(* Logix 5000 project; controller cal1632 1756-L62 rev 16.20; software revision 16.05; part 57 of 61 *)
(* tags used below, declared in another part *)
   FAULT : BOOL;
   HMI : BOOL;
   p01r09_pb_global_reset : BOOL;
   p29_di_wdr_turret : acs800_di_normal;
   p29r15_wdra_active : BOOL;
   p29r16_wdrb_active : BOOL;
   p29r20 : routine;
   p29r20_timer_warning : TIMER[4];
   p30_di_pin_1 : BOOL;
   p30_di_pin_2 : BOOL;
   p30_di_pin_3 : BOOL;
   p30_di_pin_4 : BOOL;
   p30_di_pin_5 : BOOL;
   p30_di_pin_6 : BOOL;
   p30_di_pin_7 : BOOL;
   p30_di_pin_8 : BOOL;
   p30_di_retraction_down_ls : BOOL;
   p30_di_retraction_up_ls : BOOL;
   p30_di_rotation_fault : BOOL;
   p30_di_ss_close : BOOL;
   p30_di_ss_open : BOOL;
   p30_dint_to_hmi : DINT[16];
   p30_do_retract_motion : BOOL;
   p30_do_rotation_fwd : BOOL;
   p30_do_rotation_rev : BOOL;
   p30r01 : routine;
   p30r02 : routine;
   p30r02_fault_exists : BOOL;
   p30r02_timer_fault : TIMER[4];
   p30r02_timer_warning : TIMER[4];
   p30r02_unack_fault : BOOL;
   p30r02_unack_warning : BOOL;
   p30r02_warning_exists : BOOL;
   p30r03 : routine;
   p30r03_timer_fault : TIMER[4];
   p30r03_timer_warning : TIMER[4];
   p30r04 : routine;
   p30r04_timer_fault : TIMER[4];
   p30r04_timer_warning : TIMER[4];
   p30r05 : routine;
   p30r05_timer_fault : TIMER[4];
   p30r05_timer_warning : TIMER[4];
   p30r06 : routine;
   p30r07 : routine;
   p30r08 : routine;
   p30r09 : routine;
   p30r10 : routine;
   RETACTION_DELAY_TIMER : TIMER;
   RETRACTION_DELAY_TIMER_2 : TIMER;
(* P29_Winder, continued *)

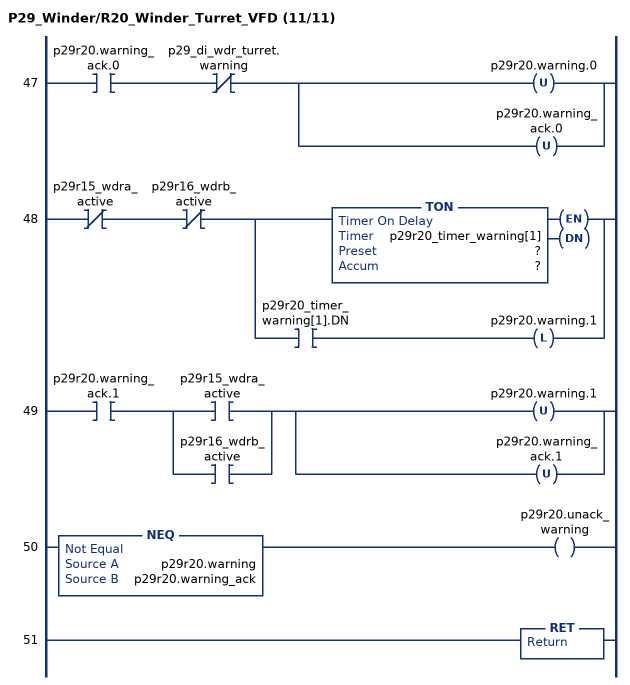
   [picture p1161: P29_Winder/R20_Winder_Turret_VFD rungs 47-51]
   47: XIC(p29r20.warning_ack.0)XIO(p29_di_wdr_turret.warning)[OTU(p29r20.warning.0) ,OTU(p29r20.warning_ack.0) ];
   48: XIO(p29r15_wdra_active)XIO(p29r16_wdrb_active)[TON(p29r20_timer_warning[1],?,?) ,XIC(p29r20_timer_warning[1].DN) OTL(p29r20.warning.1) ];
   49: XIC(p29r20.warning_ack.1)[XIC(p29r15_wdra_active) ,XIC(p29r16_wdrb_active) ][OTU(p29r20.warning.1) ,OTU(p29r20.warning_ack.1) ];
   50: NEQ(p29r20.warning,p29r20.warning_ack)OTE(p29r20.unack_warning);
   51: RET();
END_ROUTINE
END_PROGRAM

PROGRAM P30_Retraction_System   (* main routine R01_Main *)

ROUTINE R01_Main   (* ladder *)
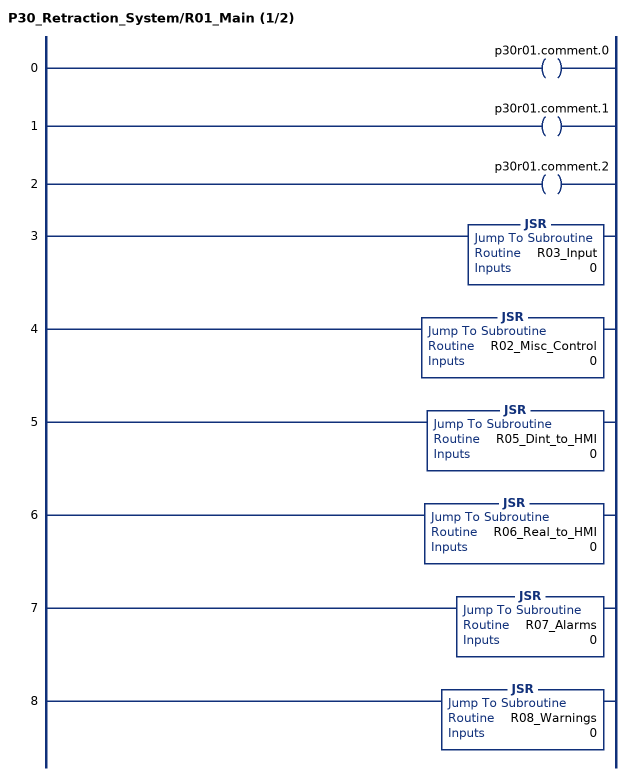
   0: OTE(p30r01.comment.0);
   1: OTE(p30r01.comment.1);
   2: OTE(p30r01.comment.2);
   3: JSR(R03_Input,0);
   4: JSR(R02_Misc_Control,0);
   5: JSR(R05_Dint_to_HMI,0);
   6: JSR(R06_Real_to_HMI,0);
   7: JSR(R07_Alarms,0);
   8: JSR(R08_Warnings,0);
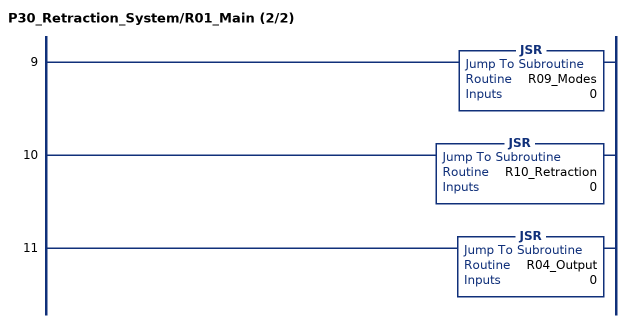
   9: JSR(R09_Modes,0);
   10: JSR(R10_Retraction,0);
   11: JSR(R04_Output,0);
END_ROUTINE

ROUTINE R02_Misc_Control   (* ladder *)
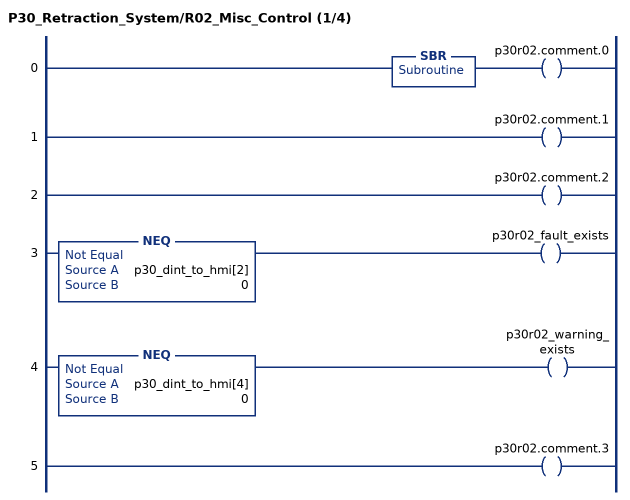
   0: SBR()OTE(p30r02.comment.0);
   1: OTE(p30r02.comment.1);
   2: OTE(p30r02.comment.2);
   3: NEQ(p30_dint_to_hmi[2],0)OTE(p30r02_fault_exists);
   4: NEQ(p30_dint_to_hmi[4],0)OTE(p30r02_warning_exists);
   5: OTE(p30r02.comment.3);
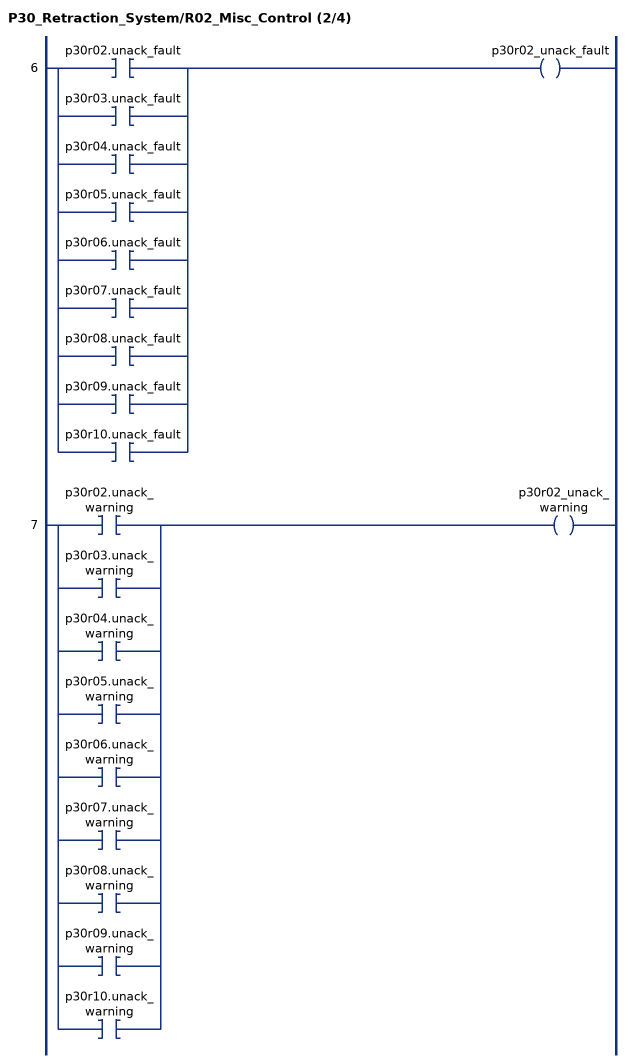
   6: [XIC(p30r02.unack_fault) ,XIC(p30r03.unack_fault) ,XIC(p30r04.unack_fault) ,XIC(p30r05.unack_fault) ,XIC(p30r06.unack_fault) ,XIC(p30r07.unack_fault) ,XIC(p30r08.unack_fault) ,XIC(p30r09.unack_fault) ,XIC(p30r10.unack_fault) ]OTE(p30r02_unack_fault);
   7: [XIC(p30r02.unack_warning) ,XIC(p30r03.unack_warning) ,XIC(p30r04.unack_warning) ,XIC(p30r05.unack_warning) ,XIC(p30r06.unack_warning) ,XIC(p30r07.unack_warning) ,XIC(p30r08.unack_warning) ,XIC(p30r09.unack_warning) ,XIC(p30r10.unack_warning) ]OTE(p30r02_unack_warning);
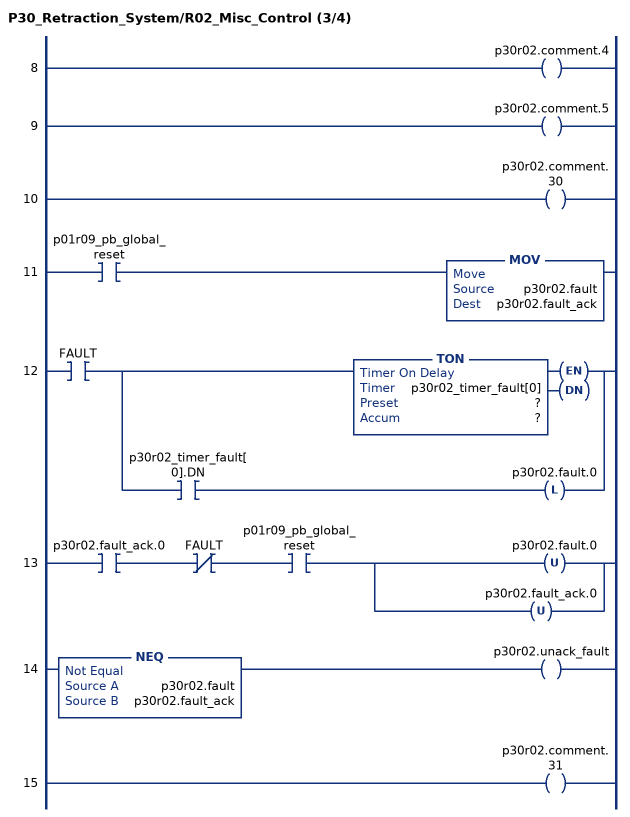
   8: OTE(p30r02.comment.4);
   9: OTE(p30r02.comment.5);
   10: OTE(p30r02.comment.30);
   11: XIC(p01r09_pb_global_reset)MOV(p30r02.fault,p30r02.fault_ack);
   12: XIC(FAULT)[TON(p30r02_timer_fault[0],?,?) ,XIC(p30r02_timer_fault[0].DN) OTL(p30r02.fault.0) ];
   13: XIC(p30r02.fault_ack.0)XIO(FAULT)XIC(p01r09_pb_global_reset)[OTU(p30r02.fault.0) ,OTU(p30r02.fault_ack.0) ];
   14: NEQ(p30r02.fault,p30r02.fault_ack)OTE(p30r02.unack_fault);
   15: OTE(p30r02.comment.31);
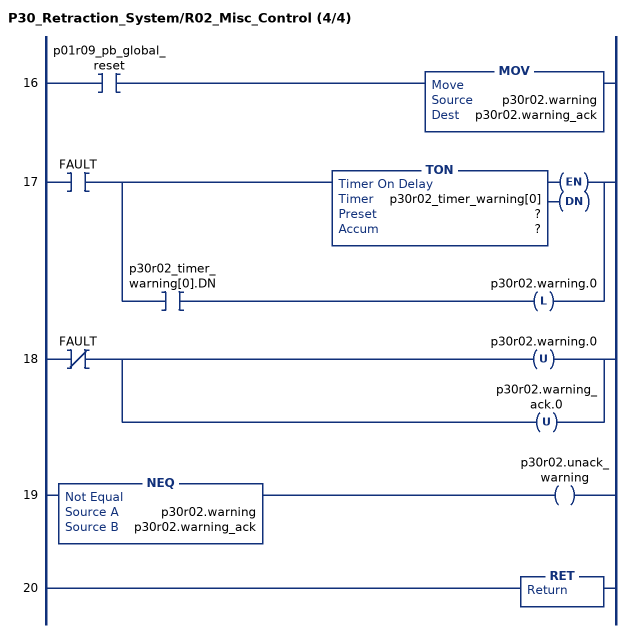
   16: XIC(p01r09_pb_global_reset)MOV(p30r02.warning,p30r02.warning_ack);
   17: XIC(FAULT)[TON(p30r02_timer_warning[0],?,?) ,XIC(p30r02_timer_warning[0].DN) OTL(p30r02.warning.0) ];
   18: XIO(FAULT)[OTU(p30r02.warning.0) ,OTU(p30r02.warning_ack.0) ];
   19: NEQ(p30r02.warning,p30r02.warning_ack)OTE(p30r02.unack_warning);
   20: RET();
END_ROUTINE

ROUTINE R03_Input   (* ladder *)
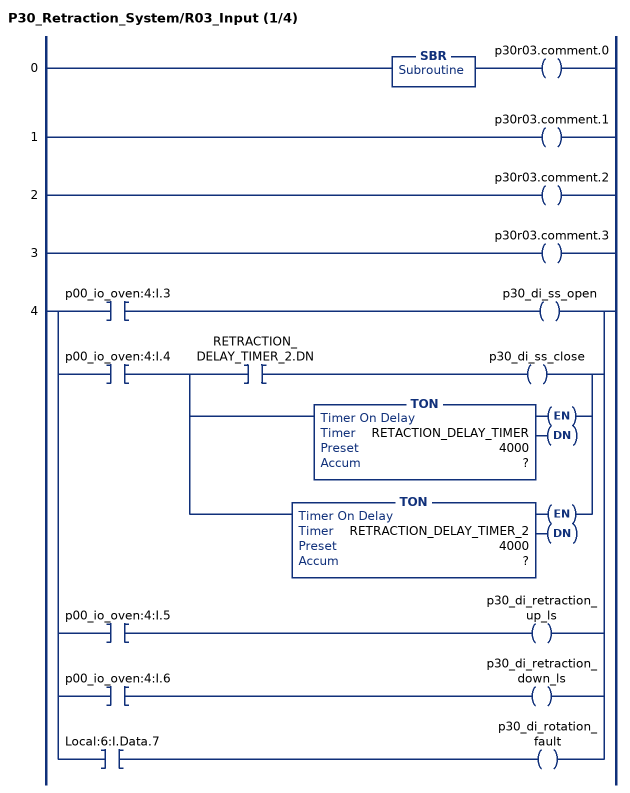
   0: SBR()OTE(p30r03.comment.0);
   1: OTE(p30r03.comment.1);
   2: OTE(p30r03.comment.2);
   3: OTE(p30r03.comment.3);
   4: [XIC(p00_io_oven:4:I.3) OTE(p30_di_ss_open) ,XIC(p00_io_oven:4:I.4) [XIC(RETRACTION_DELAY_TIMER_2.DN) OTE(p30_di_ss_close) ,TON(RETACTION_DELAY_TIMER,?,?) ,TON(RETRACTION_DELAY_TIMER_2,?,?) ] ,XIC(p00_io_oven:4:I.5) OTE(p30_di_retraction_up_ls) ,XIC(p00_io_oven:4:I.6) OTE(p30_di_retraction_down_ls) ,XIC(Local:6:I.Data.7) OTE(p30_di_rotation_fault) ];
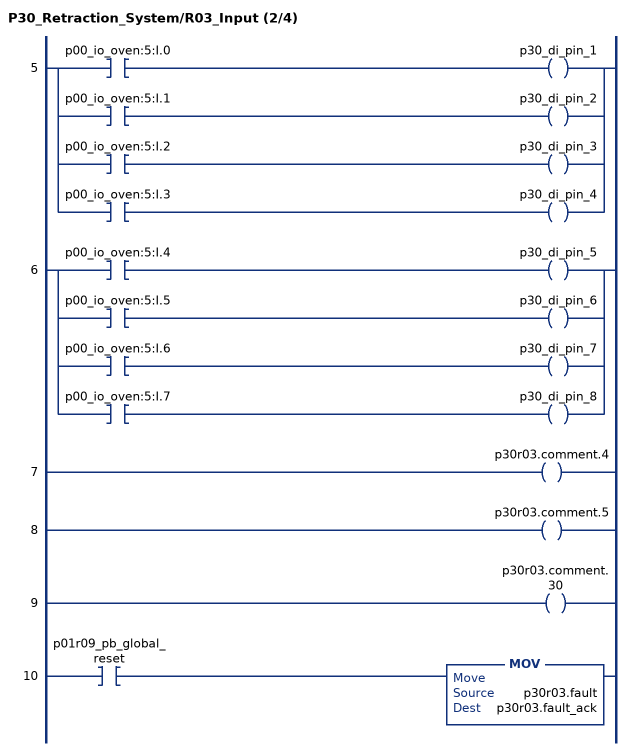
   5: [XIC(p00_io_oven:5:I.0) OTE(p30_di_pin_1) ,XIC(p00_io_oven:5:I.1) OTE(p30_di_pin_2) ,XIC(p00_io_oven:5:I.2) OTE(p30_di_pin_3) ,XIC(p00_io_oven:5:I.3) OTE(p30_di_pin_4) ];
   6: [XIC(p00_io_oven:5:I.4) OTE(p30_di_pin_5) ,XIC(p00_io_oven:5:I.5) OTE(p30_di_pin_6) ,XIC(p00_io_oven:5:I.6) OTE(p30_di_pin_7) ,XIC(p00_io_oven:5:I.7) OTE(p30_di_pin_8) ];
   7: OTE(p30r03.comment.4);
   8: OTE(p30r03.comment.5);
   9: OTE(p30r03.comment.30);
   10: XIC(p01r09_pb_global_reset)MOV(p30r03.fault,p30r03.fault_ack);
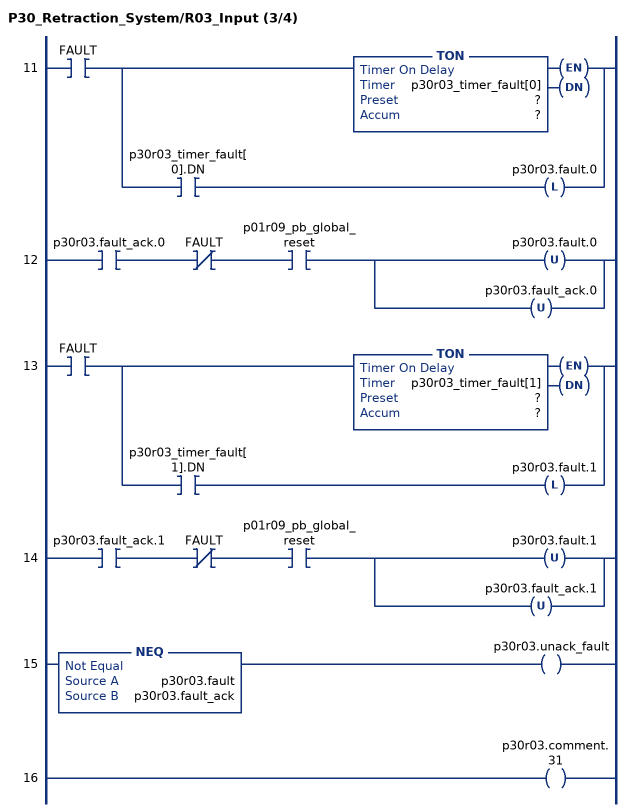
   11: XIC(FAULT)[TON(p30r03_timer_fault[0],?,?) ,XIC(p30r03_timer_fault[0].DN) OTL(p30r03.fault.0) ];
   12: XIC(p30r03.fault_ack.0)XIO(FAULT)XIC(p01r09_pb_global_reset)[OTU(p30r03.fault.0) ,OTU(p30r03.fault_ack.0) ];
   13: XIC(FAULT)[TON(p30r03_timer_fault[1],?,?) ,XIC(p30r03_timer_fault[1].DN) OTL(p30r03.fault.1) ];
   14: XIC(p30r03.fault_ack.1)XIO(FAULT)XIC(p01r09_pb_global_reset)[OTU(p30r03.fault.1) ,OTU(p30r03.fault_ack.1) ];
   15: NEQ(p30r03.fault,p30r03.fault_ack)OTE(p30r03.unack_fault);
   16: OTE(p30r03.comment.31);
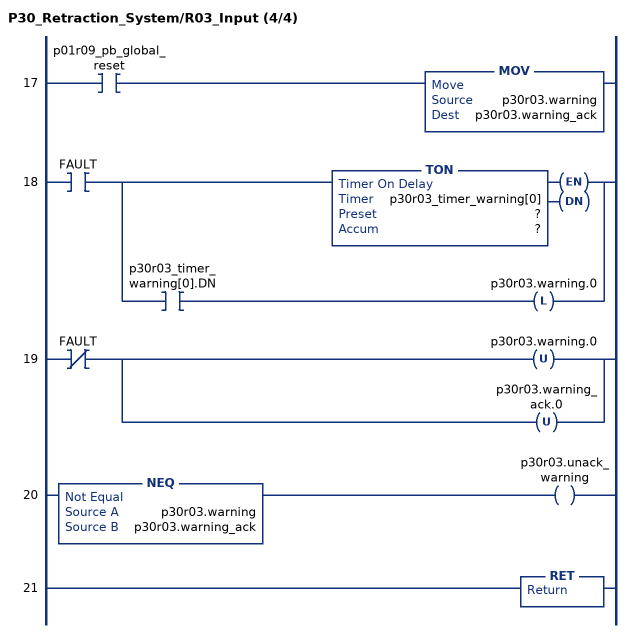
   17: XIC(p01r09_pb_global_reset)MOV(p30r03.warning,p30r03.warning_ack);
   18: XIC(FAULT)[TON(p30r03_timer_warning[0],?,?) ,XIC(p30r03_timer_warning[0].DN) OTL(p30r03.warning.0) ];
   19: XIO(FAULT)[OTU(p30r03.warning.0) ,OTU(p30r03.warning_ack.0) ];
   20: NEQ(p30r03.warning,p30r03.warning_ack)OTE(p30r03.unack_warning);
   21: RET();
END_ROUTINE

ROUTINE R04_Output   (* ladder *)
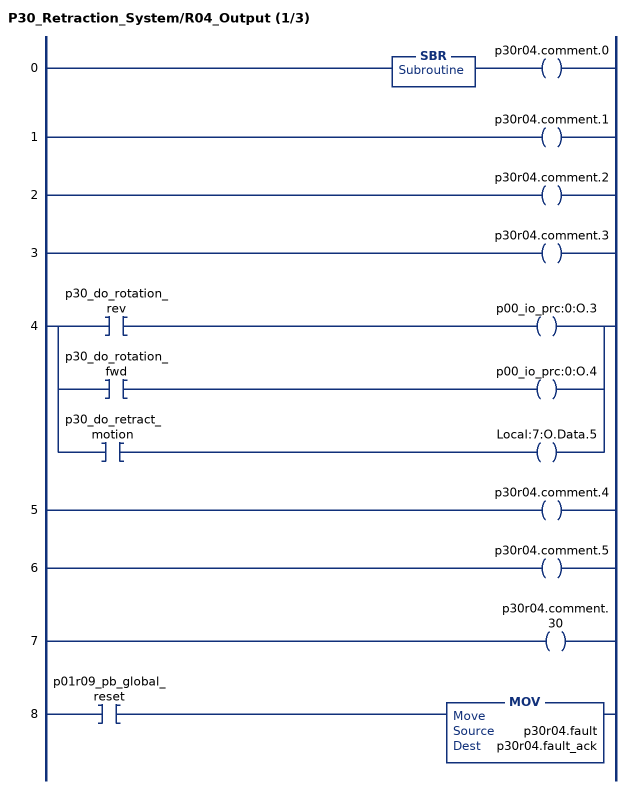
   0: SBR()OTE(p30r04.comment.0);
   1: OTE(p30r04.comment.1);
   2: OTE(p30r04.comment.2);
   3: OTE(p30r04.comment.3);
   4: [XIC(p30_do_rotation_rev) OTE(p00_io_prc:0:O.3) ,XIC(p30_do_rotation_fwd) OTE(p00_io_prc:0:O.4) ,XIC(p30_do_retract_motion) OTE(Local:7:O.Data.5) ];
   5: OTE(p30r04.comment.4);
   6: OTE(p30r04.comment.5);
   7: OTE(p30r04.comment.30);
   8: XIC(p01r09_pb_global_reset)MOV(p30r04.fault,p30r04.fault_ack);
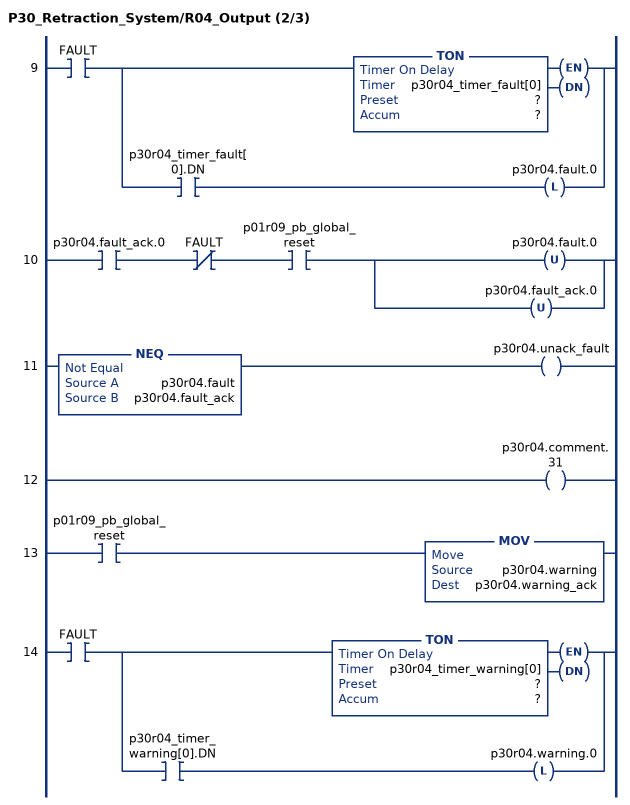
   9: XIC(FAULT)[TON(p30r04_timer_fault[0],?,?) ,XIC(p30r04_timer_fault[0].DN) OTL(p30r04.fault.0) ];
   10: XIC(p30r04.fault_ack.0)XIO(FAULT)XIC(p01r09_pb_global_reset)[OTU(p30r04.fault.0) ,OTU(p30r04.fault_ack.0) ];
   11: NEQ(p30r04.fault,p30r04.fault_ack)OTE(p30r04.unack_fault);
   12: OTE(p30r04.comment.31);
   13: XIC(p01r09_pb_global_reset)MOV(p30r04.warning,p30r04.warning_ack);
   14: XIC(FAULT)[TON(p30r04_timer_warning[0],?,?) ,XIC(p30r04_timer_warning[0].DN) OTL(p30r04.warning.0) ];
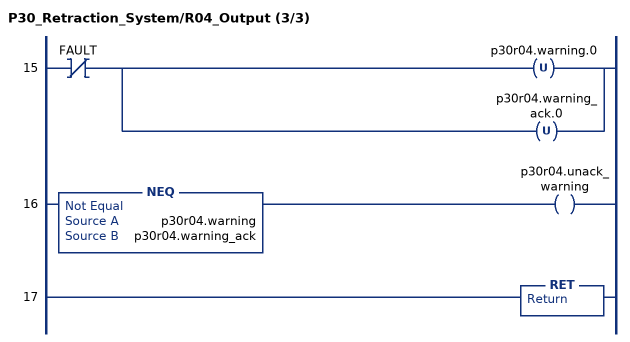
   15: XIO(FAULT)[OTU(p30r04.warning.0) ,OTU(p30r04.warning_ack.0) ];
   16: NEQ(p30r04.warning,p30r04.warning_ack)OTE(p30r04.unack_warning);
   17: RET();
END_ROUTINE

ROUTINE R05_Dint_to_HMI   (* ladder *)
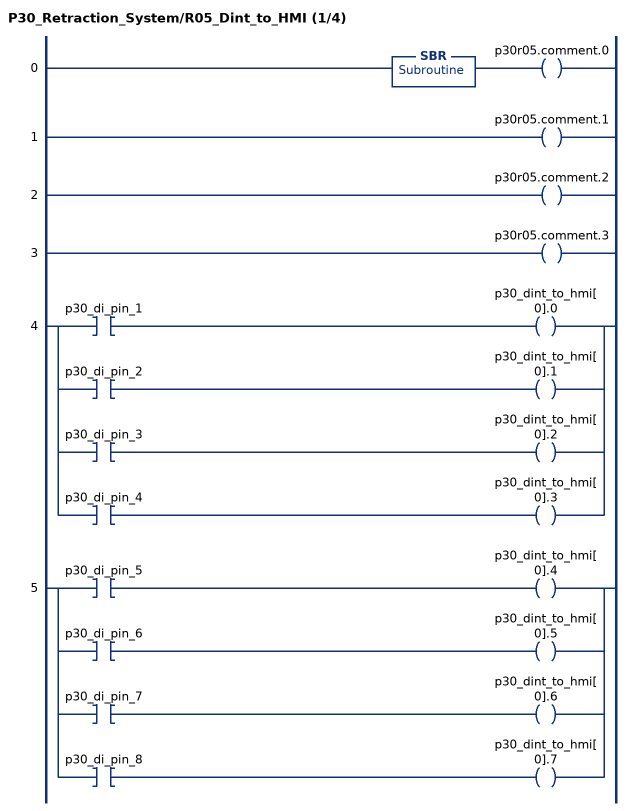
   0: SBR()OTE(p30r05.comment.0);
   1: OTE(p30r05.comment.1);
   2: OTE(p30r05.comment.2);
   3: OTE(p30r05.comment.3);
   4: [XIC(p30_di_pin_1) OTE(p30_dint_to_hmi[0].0) ,XIC(p30_di_pin_2) OTE(p30_dint_to_hmi[0].1) ,XIC(p30_di_pin_3) OTE(p30_dint_to_hmi[0].2) ,XIC(p30_di_pin_4) OTE(p30_dint_to_hmi[0].3) ];
   5: [XIC(p30_di_pin_5) OTE(p30_dint_to_hmi[0].4) ,XIC(p30_di_pin_6) OTE(p30_dint_to_hmi[0].5) ,XIC(p30_di_pin_7) OTE(p30_dint_to_hmi[0].6) ,XIC(p30_di_pin_8) OTE(p30_dint_to_hmi[0].7) ];
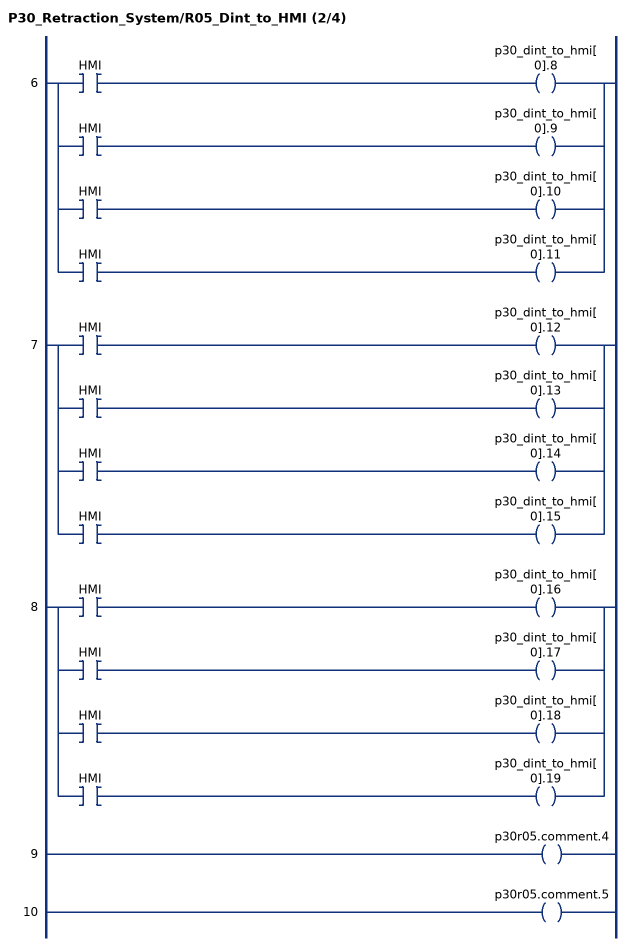
   6: [XIC(HMI) OTE(p30_dint_to_hmi[0].8) ,XIC(HMI) OTE(p30_dint_to_hmi[0].9) ,XIC(HMI) OTE(p30_dint_to_hmi[0].10) ,XIC(HMI) OTE(p30_dint_to_hmi[0].11) ];
   7: [XIC(HMI) OTE(p30_dint_to_hmi[0].12) ,XIC(HMI) OTE(p30_dint_to_hmi[0].13) ,XIC(HMI) OTE(p30_dint_to_hmi[0].14) ,XIC(HMI) OTE(p30_dint_to_hmi[0].15) ];
   8: [XIC(HMI) OTE(p30_dint_to_hmi[0].16) ,XIC(HMI) OTE(p30_dint_to_hmi[0].17) ,XIC(HMI) OTE(p30_dint_to_hmi[0].18) ,XIC(HMI) OTE(p30_dint_to_hmi[0].19) ];
   9: OTE(p30r05.comment.4);
   10: OTE(p30r05.comment.5);
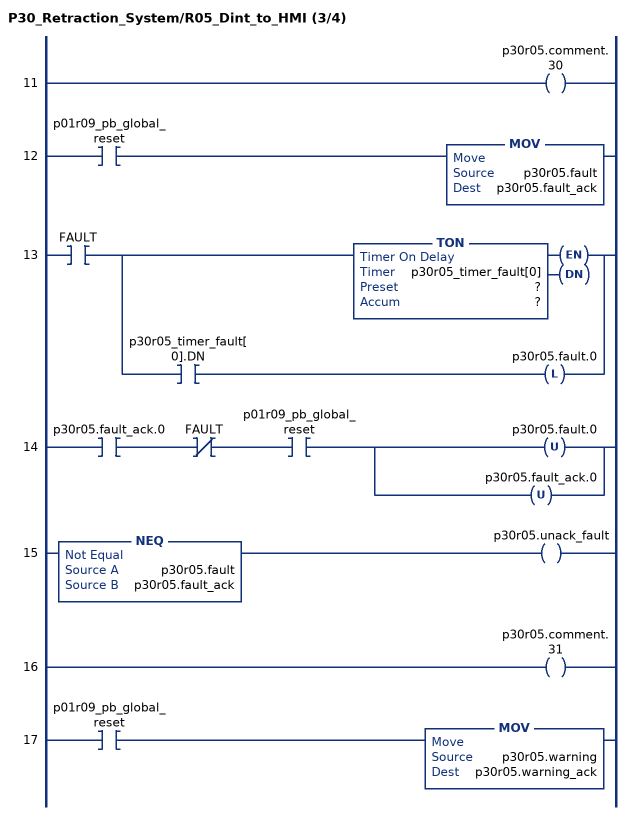
   11: OTE(p30r05.comment.30);
   12: XIC(p01r09_pb_global_reset)MOV(p30r05.fault,p30r05.fault_ack);
   13: XIC(FAULT)[TON(p30r05_timer_fault[0],?,?) ,XIC(p30r05_timer_fault[0].DN) OTL(p30r05.fault.0) ];
   14: XIC(p30r05.fault_ack.0)XIO(FAULT)XIC(p01r09_pb_global_reset)[OTU(p30r05.fault.0) ,OTU(p30r05.fault_ack.0) ];
   15: NEQ(p30r05.fault,p30r05.fault_ack)OTE(p30r05.unack_fault);
   16: OTE(p30r05.comment.31);
   17: XIC(p01r09_pb_global_reset)MOV(p30r05.warning,p30r05.warning_ack);
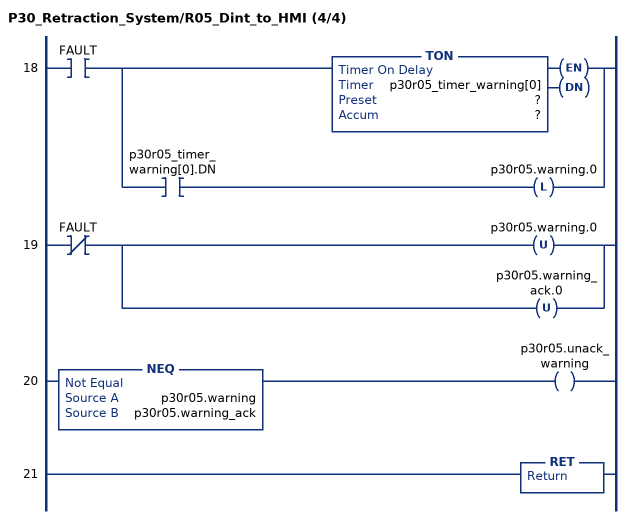
   18: XIC(FAULT)[TON(p30r05_timer_warning[0],?,?) ,XIC(p30r05_timer_warning[0].DN) OTL(p30r05.warning.0) ];
   19: XIO(FAULT)[OTU(p30r05.warning.0) ,OTU(p30r05.warning_ack.0) ];
   20: NEQ(p30r05.warning,p30r05.warning_ack)OTE(p30r05.unack_warning);
   21: RET();
END_ROUTINE
